ABB RobotStudio station: RobotStudio Workspace.rspag

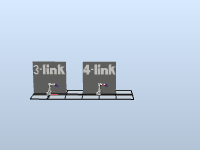
--- station ---
Station version1 (saved by RobotStudio format 3)
Controller System
  mechanical unit ROB_1: IRB120_3_58__01, 6 joints, base frame (0, 0, 0) mm
  mechanical unit ROB_2: IRB120_3_58__01_2, 6 joints, base frame (3000, 0, 0) mm
Layout (positions relative to the parent item):
  - IRB120_3_58__01 [mechanism, from Robots\IRB120_3_58_G_01.rslib] at (0, 0, 0) mm; joint values [0, 0, 0, 0, 0.5236, 0] (rad or m)
  - IRB120_3_58__01_2 [mechanism, from Robots\IRB120_3_58_G_01.rslib] at (3000, 0, 0) mm; joint values [0, 0, 0, 0, 0.5236, 0] (rad or m)
  - MyNewTool [mechanism, from Libraries\Tool_1rslib.rslib] at (364.35, 0, 594) mm, rotated rx 180 ry 60 rz 180 deg
  - MyNewTool_2 [mechanism, from Libraries\Tool_1rslib.rslib] at (3364.35, 0, 594) mm, rotated rx 180 ry 60 rz 180 deg
  - Wall [part, from Libraries\Wall.rslib] at (-1000, 150, 0) mm
  - Wall2 [part, from Libraries\Wall2.rslib] at (0, 150, 0) mm
  - 3 [part, from Libraries\3.rslib] at (-203.1, 0, 2640.47) mm, rotated rx 90 ry 0 rz 0 deg
  - 4 [part, from Libraries\4.rslib] at (2237.05, 0, 3057.64) mm, rotated rx 90 ry 0 rz 0 deg
  - hyphen [part, from Libraries\hifen.rslib] at (2501.1, 0, 1530.78) mm, rotated rx 90 ry 0 rz 0 deg
  - hyphen_2 [part, from Libraries\hifen.rslib] at (-579.72, 0, 1530.78) mm, rotated rx 90 ry 0 rz 0 deg
  - i [part, from Libraries\i.rslib] at (6.71, 0, 2650.44) mm, rotated rx 90 ry 0 rz 0 deg
  - i_2 [part, from Libraries\i.rslib] at (3065.42, 0, 2650.44) mm, rotated rx 90 ry 0 rz 0 deg
  - k [part, from Libraries\k.rslib] at (0, 0, 2646.78) mm, rotated rx 90 ry 0 rz 0 deg
  - k_2 [part, from Libraries\k.rslib] at (3032.61, 0, 2646.78) mm, rotated rx 90 ry 0 rz 0 deg
  - l [part, from Libraries\l.rslib] at (-369.34, 0, 1257.2) mm, rotated rx 90 ry 0 rz 0 deg
  - l_2 [part, from Libraries\l.rslib] at (2704.62, 0, 1257.2) mm, rotated rx 90 ry 0 rz 0 deg
  - n [part, from Libraries\n.rslib] at (0, 0, 2647.94) mm, rotated rx 90 ry 0 rz 0 deg
  - n_2 [part, from Libraries\n.rslib] at (3053.54, 0, 2647.94) mm, rotated rx 90 ry 0 rz 0 deg
Attachment: MyNewTool is attached to IRB120_3_58__01 / Link6
Attachment: MyNewTool_2 is attached to IRB120_3_58__01_2 / Link6
Targets, tools, work objects and paths stored in the station and not in the controller backup, written as RAPID:
! task T_ROB1
MODULE Action
  VAR jointtarget joints:=[[0,0,0,0,0,0],[9E9,9E9,9E9,9E9,9E9,9E9]];
ENDMODULE

! task T_ROB2
MODULE Action2
  VAR jointtarget joints:=[[0,0,0,0,0,0],[9E9,9E9,9E9,9E9,9E9,9E9]];
ENDMODULE


--- Backups/System/RAPID/TASK1/PROGMOD/Action.mod ---
MODULE Action
    VAR num n_link;
    VAR num n_times;
    VAR num J1{100};
    VAR num J2{100};
    VAR num J3{100};
    VAR num J4{100};
    VAR num J5{100};
    VAR num J6{100};
    VAR num var2;
    VAR num var3;
    VAR num var5;
    VAR pos CPosition;
    VAR string position_str;
    VAR string anglesr;
    VAR jointtarget joints;


    PROC ReadingArm()
        VAR string filelocation:="arm.txt";
        VAR iodev file;
        Open filelocation,file\Read;
        n_link:=ReadNum(file\Delim:="\10");
        J1{1}:=0;
        var2:=ReadNum(file\Delim:="\10");
        J2{1}:=var2;
        var3:=ReadNum(file\Delim:="\10");
        J3{1}:=var3;
        J4{1}:=0;
        var5:=ReadNum(file);
        J5{1}:=var5;
        J6{1}:=0;
        Close file;
    ENDPROC

    PROC ReadingAng()
        VAR string filelocation:="angles.txt";
        VAR iodev file;
        Open filelocation,file\Read;
        n_times:=ReadNum(file\Delim:="\10");
        FOR count FROM 2 TO n_times+1 DO
            J1{count}:=0;
            var2:=var2+ReadNum(file\Delim:=",");
            J2{count}:=var2;
            var3:=var3+ReadNum(file\Delim:=",");
            J3{count}:=var3;
            J4{count}:=0;
            var5:=var5+ReadNum(file);
            J5{count}:=var5;
            J6{count}:=0;
        ENDFOR
        Close file;
    ENDPROC

    !a method for the the pos
    PROC pWriteSomething()
        VAR string filelocation:="out.txt";
        VAR iodev file;
        Open filelocation,file\Append;
        position_str:=NumToStr(CPosition.x,3)+","+
NumToStr(CPosition.y,3)+","+NumToStr(CPosition.z,3);
        Write file,position_str;
        Close file;
    ENDPROC

    !a method for checking the angles
    PROC WI()
        VAR string location:="wi.txt";
        VAR iodev filea;
        Open location,filea\Append;
        FOR count FROM 1 TO n_times+1 DO
            anglesr:=NumToStr(J2{count},3)+","+
NumToStr(J3{count},3)+","+NumToStr(J5{count},3);
            Write filea,anglesr;
        ENDFOR
        Close filea;

    ENDPROC

    PROC main()
        ReadingArm;
        IF n_link=3 THEN
            ReadingAng;
            WI;
            FOR count FROM 1 TO n_times+1 DO
                joints.robax.rax_1:=J1{count};
                joints.robax.rax_2:=J2{count};
                joints.robax.rax_3:=J3{count};
                joints.robax.rax_4:=J4{count};
                joints.robax.rax_5:=J5{count};
                joints.robax.rax_6:=J6{count};
                MoveAbsJ joints,v1000,fine,Tool_1\WObj:=wobj0;
                CPosition:=CPos();
                pWriteSomething;
            ENDFOR
        ENDIF
    ENDPROC
ENDMODULE

--- Backups/System/RAPID/TASK1/PROGMOD/CalibData.mod ---
MODULE CalibData
	PERS tooldata Tool_1:=[TRUE,[[0,150,105],[1,0,0,0]],[1,[0,0,1],[1,0,0,0],0,0,0]];
ENDMODULE

--- Backups/System/RAPID/TASK1/SYSMOD/LINKEDM.sys ---
%%%
  VERSION:1
  LANGUAGE:ENGLISH
%%%

MODULE LINKEDM (SYSMODULE)

! FOLLOWER
!     Name of electronically linked follower axis used by operator at teach pendent.
      PERS string l_f_axis_name{5}       :=  ["",  "", "", "", ""];

!     Name of the mechanical unit for follower axis.
      PERS string l_f_mecunt_n{5}  :=  ["", "", "", "", ""];

!     Linked follower axis number in the mechanical unit (first axis in mech. unit is number 1).
      PERS num l_f_axis_no{5}      :=  [0,          0,   0,  0,  0];

! MASTER
!     Name of the mechanical unit for linked master axis.
      PERS string l_m_mecunt_n{5} :=  ["", "", "", "", ""];

!     Linked master axis number in the mechanical unit (first axis in mech. unit is number 1).
!     See axis number table in documentation for different master mechanical units.
      PERS num l_m_axis_no{5}     :=  [0,  0,  0,  0,  0];

! POSITION OFFSET
!     The increase of the allowed offset position between the master and follower
!     positions, used when starting AUTO mode. As soon as the offset is decreased
!     the old configurated parameter is used.
!     Example: 3 => the configurated value of allowed offset is increased 3 times.
      PERS num offset_ratio{5}       :=  [10,  10,   10,  10,  10];

! SPEED RATIO
!     Speed_ratio used in AUTO and JOG modes [ very_slow   slow    normal    fast]
!     Value 1 = max allowed manual speed.
      CONST num speed_ratio {20}      := [0.01, 0.01, 0.01, 0.01, 0.01,
                                          0.05, 0.05, 0.05, 0.05, 0.05,
                                          0.20, 0.20, 0.20, 0.20, 0.20,
                                          1.00, 1.00, 1.00, 1.00, 1.00];

! STEP SIZE
!     Displacement position used in JOG mode for each activation of positive or
!     negative movement.                  [very_short    short   normal   long]
!     Unit degees or meter.
      CONST num displacement {20}     := [0.001, 0.001, 0.001, 0.001, 0.001,
                                          0.005, 0.005, 0.005, 0.005, 0.005,
                                          0.020, 0.020, 0.020, 0.020, 0.020,
                                          0.100, 0.100, 0.100, 0.100, 0.100];


!-------------------------------------------------------------
 PROC Linked_m ()
      Linked_m_exe ;
 ENDPROC
ENDMODULE

--- Backups/System/RAPID/TASK2/PROGMOD/Action2.mod ---
MODULE Action2
    VAR num n_link;
    VAR num n_times;
    VAR num J1{100};
    VAR num J2{100};
    VAR num J3{100};
    VAR num J4{100};
    VAR num J5{100};
    VAR num J6{100};
    VAR num var2;
    VAR num var3;
    VAR num var5;
    VAR pos CPosition;
    VAR string position_str;
    VAR string anglesr;
    VAR jointtarget joints;


    PROC ReadingArm()
        VAR string filelocation:="arm.txt";
        VAR iodev file;
        Open filelocation,file\Read;
        n_link:=ReadNum(file\Delim:="\10");
        J1{1}:=0;
        var2:=ReadNum(file\Delim:="\10");
        J2{1}:=var2;
        var3:=ReadNum(file\Delim:="\10");
        J3{1}:=var3;
        J4{1}:=0;
        var5:=ReadNum(file);
        J5{1}:=var5;
        J6{1}:=0;
        Close file;
    ENDPROC

    PROC ReadingAng()
        VAR string filelocation:="angles.txt";
        VAR iodev file;
        Open filelocation,file\Read;
        n_times:=ReadNum(file\Delim:="\10");
        FOR count FROM 2 TO n_times+1 DO
            J1{count}:=0;
            var2:=var2+ReadNum(file\Delim:=",");
            J2{count}:=var2;
            var3:=var3+ReadNum(file\Delim:=",");
            J3{count}:=var3;
            J4{count}:=0;
            var5:=var5+ReadNum(file);
            J5{count}:=var5;
            J6{count}:=0;
        ENDFOR
        Close file;
    ENDPROC

    !a method for the the pos
    PROC pWriteSomething()
        VAR string filelocation:="out.txt";
        VAR iodev file;
        Open filelocation,file\Append;
        position_str:=NumToStr(CPosition.x,3)+","+
NumToStr(CPosition.y,3)+","+NumToStr(CPosition.z,3);
        Write file,position_str;
        Close file;
    ENDPROC

    !a method for checking the angles
    PROC WI()
        VAR string location:="wi.txt";
        VAR iodev filea;
        Open location,filea\Append;
        FOR count FROM 1 TO n_times+1 DO
            anglesr:=NumToStr(J2{count},3)+","+
NumToStr(J3{count},3)+","+NumToStr(J5{count},3);
            Write filea,anglesr;
        ENDFOR
        Close filea;

    ENDPROC

    PROC main()
        ReadingArm;
        IF n_link=4 THEN
            ReadingAng;
            WI;
            FOR count FROM 1 TO n_times+1 DO
                joints.robax.rax_1:=J1{count};
                joints.robax.rax_2:=J2{count};
                joints.robax.rax_3:=J3{count};
                joints.robax.rax_4:=J4{count};
                joints.robax.rax_5:=J5{count};
                joints.robax.rax_6:=J6{count};
                MoveAbsJ joints,v1000,fine,Tool_1\WObj:=wobj0;
                CPosition:=CPos();
                pWriteSomething;
            ENDFOR
        ENDIF
    ENDPROC
ENDMODULE
